// TIA Portal project "2022.06.05_上升下降沿" (V17)

(* hardware
DEVICE "S7-1200 station_1"  S7-1200 Station
   slot 0: "Rack_0"  S7-1200 Rack  Rack  V1.0
   slot 1: "PLC_1"  CPU 1212C DC/DC/DC  6ES7 212-1AE40-0XB0  V4.5
*)

// ===== PLC "PLC_1"  CPU 1212C DC/DC/DC =====

VAR_GLOBAL   // PLC tag table "默认变量表"
   "Tag_1" AT %I0.0 : Bool;
   "自动复位" AT %M0.0 : Bool;
   "故障" AT %I0.2 : Bool;
   "Tag_4" AT %MW10 : Int;
   "Tag_5" AT %Q0.0 : Bool;
   "手动复位" AT %I0.1 : Bool;
   "初始位" AT %M1.0 : Bool;
   "Tag_2" AT %M0.1 : Bool;
   "赋值" AT %I0.3 : Bool;
   "Tag_7" AT %I0.4 : Bool;
   "加" AT %I0.5 : Bool;
   "Tag_9" AT %M10.0 : Bool;
   "减" AT %I0.6 : Bool;
   "手动复位(1)" AT %I0.7 : Bool;
   "Tag_12" AT %M10.1 : Bool;
   "当前值" AT %MW20 : Int;
   "Tag_6" AT %M0.2 : Bool;
   "5次" AT %M0.3 : Bool;
   "运行电机" AT %Q0.1 : Bool;
   "备用电机" AT %Q0.2 : Bool;
END_VAR

// folder: System blocks/Program resources

DATA_BLOCK "IEC_Counter_0_DB"   // DB1
{ S7_Optimized_Access := 'TRUE' }
AUTHOR : Simatic
FAMILY : IEC
NAME : CNTR
VERSION : 1.0
// stored: InstanceOfName IEC_COUNTER
"IEC_COUNTER"
BEGIN
END_DATA_BLOCK

DATA_BLOCK "IEC_Counter_0_DB_1"   // DB2
{ S7_Optimized_Access := 'TRUE' }
AUTHOR : Simatic
FAMILY : IEC
NAME : CNTR
VERSION : 1.0
// stored: InstanceOfName IEC_COUNTER
"IEC_COUNTER"
BEGIN
END_DATA_BLOCK

DATA_BLOCK "IEC_Counter_0_DB_2"   // DB3
{ S7_Optimized_Access := 'TRUE' }
AUTHOR : Simatic
FAMILY : IEC
NAME : CNTR
VERSION : 1.0
// stored: InstanceOfName IEC_COUNTER
"IEC_COUNTER"
BEGIN
END_DATA_BLOCK

DATA_BLOCK "IEC_Timer_0_DB"   // DB4
{ S7_Optimized_Access := 'TRUE' }
AUTHOR : Simatic
FAMILY : IEC
NAME : IEC_TMR
VERSION : 1.0
// stored: InstanceOfName IEC_TIMER
"IEC_TIMER"
BEGIN
END_DATA_BLOCK

DATA_BLOCK "IEC_Counter_0_DB_3"   // DB5
{ S7_Optimized_Access := 'TRUE' }
AUTHOR : Simatic
FAMILY : IEC
NAME : CNTR
VERSION : 1.0
// stored: InstanceOfName IEC_COUNTER
"IEC_COUNTER"
BEGIN
END_DATA_BLOCK

// folder: (top level)

ORGANIZATION_BLOCK "Main"   // OB1, LAD, ProgramCycle
TITLE = "Main Program Sweep (Cycle)"
{ S7_Optimized_Access := 'TRUE' }
VERSION : 0.1
   VAR_INPUT
      Initial_Call : Bool;   // Initial call of this OB
      Remanence : Bool;   // =True, if remanent data are available
   END_VAR
   VAR_TEMP   // added for the SCL form of the ladder/FBD networks
      _w1 : Bool;
      _w2 : Bool;
   END_VAR
BEGIN

REGION Network 1
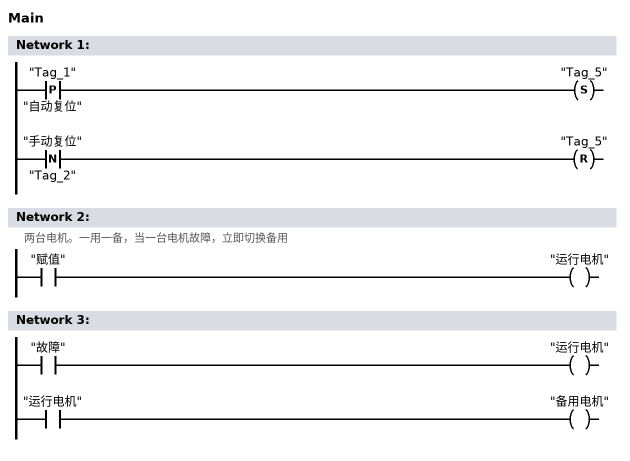
   RUNG wire#powerrail
      P_Contact(operand := "Tag_1", bit := "自动复位")
      S_Coil( "Tag_5" )
   END_RUNG
   RUNG wire#powerrail
      N_Contact(operand := "手动复位", bit := "Tag_2")
      R_Coil( "Tag_5" )
   END_RUNG
   // the same network as SCL:
   #_w1 := "Tag_1" AND NOT "自动复位";   // rising edge of "Tag_1"
   "自动复位" := "Tag_1";
   IF #_w1 THEN "Tag_5" := TRUE; END_IF;
   #_w2 := NOT "手动复位" AND "Tag_2";   // falling edge of "手动复位"
   "Tag_2" := "手动复位";
   IF #_w2 THEN "Tag_5" := FALSE; END_IF;
END_REGION

REGION Network 2
   // 两台电机。一用一备，当一台电机故障，立即切换备用
   RUNG wire#powerrail
      Contact( "赋值" )
      Coil( "运行电机" )
   END_RUNG
   // the same network as SCL:
   "运行电机" := "赋值";
END_REGION

REGION Network 3
   RUNG wire#powerrail
      Contact( "故障" )
      Coil( "运行电机" )
   END_RUNG
   RUNG wire#powerrail
      Contact( "运行电机" )
      Coil( "备用电机" )
   END_RUNG
   // the same network as SCL:
   "运行电机" := "故障";
   "备用电机" := "运行电机";
END_REGION
END_ORGANIZATION_BLOCK